FUNCTION Convert_TOD_TO_INT : Hresult
VAR_INPUT
	in : TOD;
	out : REFERENCE TO INT;
END_VAR
VAR
	converted : INT;
END_VAR
VAR CONSTANT
	INCOMPATIBLE : HRESULT := 16#9811070E;
END_VAR

converted := TOD_TO_INT(in);

IF (INT_TO_TOD(converted) <> in) THEN
	Convert_TOD_TO_INT := INCOMPATIBLE;
	RETURN;
END_IF

out := converted;

END_FUNCTION

(* stored: Version 1.1.0.1, ProductVersion 3.1.4024.12
   POU Convert_TOD_TO_INT: Id {9e8a57b1-aacb-48ff-b8d5-c7efae7cb6fc}, SpecialFunc None *)
